ACTION act_Macinatore:
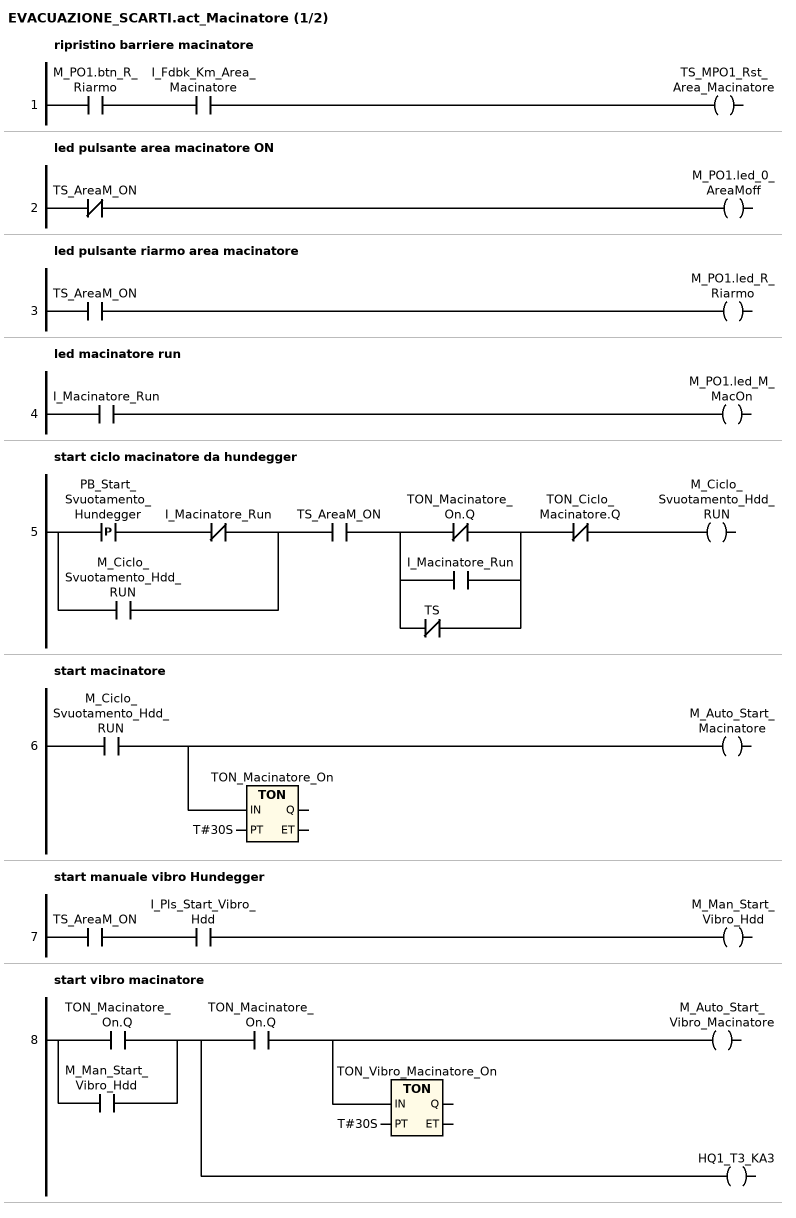
// NETWORK 1: ripristino barriere macinatore
TS_MPO1_Rst_Area_Macinatore := M_PO1.btn_R_Riarmo AND I_Fdbk_Km_Area_Macinatore;

// NETWORK 2: led pulsante area macinatore ON
M_PO1.led_0_AreaMoff := NOT TS_AreaM_ON;

// NETWORK 3: led pulsante riarmo area macinatore
M_PO1.led_R_Riarmo := TS_AreaM_ON;

// NETWORK 4: led macinatore run
M_PO1.led_M_MacOn := I_Macinatore_Run;

// NETWORK 5: start ciclo macinatore da hundegger
_rt1(CLK := PB_Start_Svuotamento_Hundegger);
M_Ciclo_Svuotamento_Hdd_RUN := (_rt1.Q AND NOT I_Macinatore_Run OR M_Ciclo_Svuotamento_Hdd_RUN) AND TS_AreaM_ON AND (NOT TON_Macinatore_On.Q OR I_Macinatore_Run OR NOT TS) AND NOT TON_Ciclo_Macinatore.Q;

// NETWORK 6: start macinatore
M_Auto_Start_Macinatore := M_Ciclo_Svuotamento_Hdd_RUN;
TON_Macinatore_On(IN := M_Ciclo_Svuotamento_Hdd_RUN, PT := T#30S); // TON

// NETWORK 7: start manuale vibro Hundegger
M_Man_Start_Vibro_Hdd := TS_AreaM_ON AND I_Pls_Start_Vibro_Hdd;

// NETWORK 8: start vibro macinatore
_w1 := TON_Macinatore_On.Q OR M_Man_Start_Vibro_Hdd;
_w2 := _w1 AND TON_Macinatore_On.Q;
M_Auto_Start_Vibro_Macinatore := _w2;
TON_Vibro_Macinatore_On(IN := _w2, PT := T#30S); // TON
HQ1_T3_KA3 := _w1;

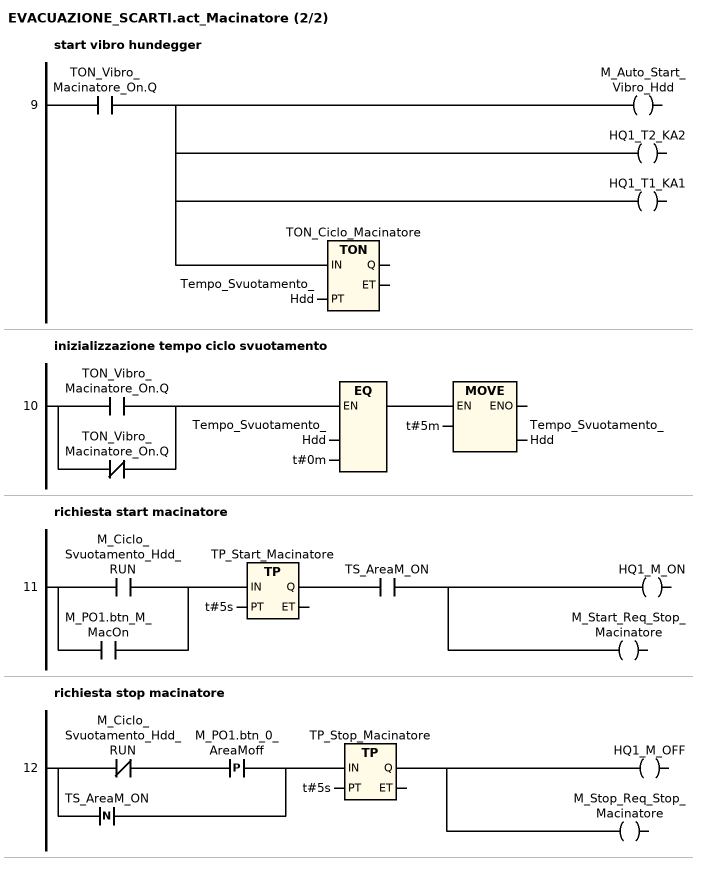
// NETWORK 9: start vibro hundegger
M_Auto_Start_Vibro_Hdd := TON_Vibro_Macinatore_On.Q;
HQ1_T2_KA2 := TON_Vibro_Macinatore_On.Q;
HQ1_T1_KA1 := TON_Vibro_Macinatore_On.Q;
TON_Ciclo_Macinatore(IN := TON_Vibro_Macinatore_On.Q, PT := Tempo_Svuotamento_Hdd); // TON

// NETWORK 10: inizializzazione tempo ciclo svuotamento
IF (TON_Vibro_Macinatore_On.Q OR NOT TON_Vibro_Macinatore_On.Q) AND Tempo_Svuotamento_Hdd = t#0m THEN
    Tempo_Svuotamento_Hdd := t#5m;
END_IF

// NETWORK 11: richiesta start macinatore
TP_Start_Macinatore(IN := M_Ciclo_Svuotamento_Hdd_RUN OR M_PO1.btn_M_MacOn, PT := t#5s); // TP
_w3 := TP_Start_Macinatore.Q AND TS_AreaM_ON;
HQ1_M_ON := _w3;
M_Start_Req_Stop_Macinatore := _w3;

// NETWORK 12: richiesta stop macinatore
_rt2(CLK := M_PO1.btn_0_AreaMoff);
_ft1(CLK := TS_AreaM_ON);
TP_Stop_Macinatore(IN := NOT M_Ciclo_Svuotamento_Hdd_RUN AND _rt2.Q OR _ft1.Q, PT := t#5s); // TP
HQ1_M_OFF := TP_Stop_Macinatore.Q;
M_Stop_Req_Stop_Macinatore := TP_Stop_Macinatore.Q;
END_ACTION

ACTION act_OUTPUT:

IF NOT bSIMULA_out THEN
	
	//TERM9 EL2008 H-Q1
	glo_dig_out_HQ1[1]		:=	Dis_Scarico_Hundegger;//S1_U1;									//DIGOUT CH1		Valvola aria pulizia ingresso M12
	glo_dig_out_HQ1[2]		:=	HQ1_T1_KA1;								//DIGOUT CH2		T1 Vibrotrasp buca
	glo_dig_out_HQ1[3]		:=	HQ1_T2_KA2;								//DIGOUT CH3		T2 Nastro elev buca
	glo_dig_out_HQ1[4]		:=	HQ1_T3_KA3;// AND NOT SensInMac;			//DIGOUT CH4		T3 Vibrotrasp macinatore
	glo_dig_out_HQ1[5]		:=	HQ1_T5M2_A_KA4;							//DIGOUT CH5		Apre scarico trasp orizz
	glo_dig_out_HQ1[6]		:=	HQ1_T5_KA5;								//DIGOUT CH6		Trasp elevat a parete
	glo_dig_out_HQ1[7]		:=	HQ1_T6_KA6;								//DIGOUT CH7		Trasp orizza a parete
	glo_dig_out_HQ1[8]		:=	HQ1_T5M2_C_KA7;							//DIGOUT CH8		Chiude scarico trasp orizz
	
	//TERM10 EL2008 H-Q1
	glo_dig_out_HQ1[9]		:= HQ1_T7_A_KA8;							//DIGOUT CH1		Caricatore macinat Avanti
	glo_dig_out_HQ1[10]		:= HQ1_T7_I_KA9;							//DIGOUT CH2		Caricatore macinat Indietro
	glo_dig_out_HQ1[11]		:= HQ1_M_ON;								//DIGOUT CH3		Macinatore ON impulsivo
	glo_dig_out_HQ1[12]		:= HQ1_M_OFF;								//DIGOUT CH4		Macinatore OFF impulsivo
	glo_dig_out_HQ1[13]		:= HQ1_T4_KA4;								//DIGOUT CH5		T4 Trasportatore silos macinatore	
	glo_dig_out_HQ1[14]		:= HQ1_S1_ValvolaStellare;					//DIGOUT CH6		Valvola stellare scarico silos 1	
	glo_dig_out_HQ1[15]		:= HQ1_RaclaON;								//DIGOUT CH7		Rancia: avviata da quadro silos
	glo_dig_out_HQ1[16]		:= HQ1_BrichettatriceON;					//DIGOUT CH8		Bricchettatrice: avviata da quadro silos

	//M_PO1											
	//IOLINK CH4		PULSANTIERA BNI005M
	glo_dig_out_T3C01[5] 	:= M_PO1.led_M_MacOn;						//BOTTONE '0'
	glo_dig_out_T3C01[8]	:= M_PO1.led_R_Riarmo;						//BOTTONE 'r'
	glo_dig_out_T3C01[6]	:= M_PO1.led_0_AreaMoff;					//TASTO 'M'
	
	//S1_PO1											
	//IOLINK CH4		PULSANTIERA BNI005M
					//BOTTONE 'r'

END_IF
END_ACTION

ACTION act_Semafori:

//#######################################################
//####################    SEMAFORI   ####################
//#######################################################

IF TS_AreaM_ON THEN
	IF I_Macinatore_Run  THEN
		fbS1_Se1(bON:= TRUE, sColore:= 3, bBlink:= TRUE, semaforo=> S1_Se1);	//verde	
	ELSE
		fbS1_Se1(bON:= TRUE, sColore:= 4, bBlink:= TRUE, semaforo=> S1_Se1);	//arancio
	END_IF
ELSE	
	fbS1_Se1(bON:= TRUE, sColore:= 2, bBlink:= TRUE, semaforo=> S1_Se1);	//rosso
END_IF
END_ACTION

ACTION act_Sensori:

//#######################################################
//####################    SENSORI   #####################
//#######################################################
//SOTTO HUNDEGGER
//CODA CIRCOLARE VALORI SENSORE inbit
T1SO1tmravg(IN:=TRUE,PT:=T#200MS);
T1SO1maxCnt:= REAL_TO_INT(T1SO1maxTimeavg*1000/200);
IF T1SO1maxCnt > 99 THEN
	T1SO1maxCnt:=99;
END_IF
IF T1SO1tmravg.Q THEN
	T1SO1tmravg(IN:=FALSE);	
	//CONTATORE TEMPO MASSIMO CAMPIONATURA
	IF T1SO1cnt < T1SO1maxCnt-1 THEN
		T1SO1cnt:=T1SO1cnt+1;	
	ELSE
		T1SO1cnt:=0;
	END_IF
	//POPOLO ARRAY LETTURE SENSORE in bit			
	T1SO1arravg[T1SO1cnt]:= T1_SO1;
END_IF
//MEDIA VALORI inbit
T1SO1cnt3:=0;
T1SO1sumavg:=0;
FOR T1SO1cnt2:=1 TO T1SO1maxCnt-1 DO
	IF T1SO1arravg[T1SO1cnt2] > 0 THEN
		T1SO1sumavg:= T1SO1sumavg + T1SO1arravg[T1SO1cnt2];
		T1SO1cnt3:=T1SO1cnt3+1;
	END_IF
END_FOR
IF T1SO1sumavg > 0 THEN
	T1SO1avg:=(T1SO1sumavg/T1SO1cnt3);	
END_IF
T1.SO1_fb(
	lettura:= REAL_TO_INT(T1SO1avg), 
	distanzaAVuoto:=6150,
	valSoglia:= solgiaT1SO1, 
	filtertime:=0,
	full=> appT1S01_Full);		
	
	//T1S01 full ritardato di 10 secondi 
	tmrT1S01_Full(IN:=appT1S01_Full,PT:=T#10S);
	T1.SO1_full := tmrT1S01_Full.Q;
	
//INGRESSO al T3
//CODA CIRCOLARE VALORI SENSORE inbit
T3S1tmravg(IN:=TRUE,PT:=T#200MS);
T3S1maxCnt:= REAL_TO_INT(T3S1maxTimeavg*1000/200);
IF T3S1maxCnt > 99 THEN
	T3S1maxCnt:=99;
END_IF
IF T3S1tmravg.Q THEN
	T3S1tmravg(IN:=FALSE);	
	//CONTATORE TEMPO MASSIMO CAMPIONATURA
	IF T3S1cnt < T3S1maxCnt-1 THEN
		T3S1cnt:=T3S1cnt+1;	
	ELSE
		T3S1cnt:=0;
	END_IF
	//POPOLO ARRAY LETTURE SENSORE in bit			
	T3S1arravg[T3S1cnt]:= T3_S1;
END_IF
//MEDIA VALORI inbit
T3S1cnt3:=0;
T3S1sumavg:=0;
FOR T3S1cnt2:=1 TO T3S1maxCnt-1 DO
	IF T3S1arravg[T3S1cnt2] > 0 THEN
		T3S1sumavg:= T3S1sumavg + T3S1arravg[T3S1cnt2];
		T3S1cnt3:=T3S1cnt3+1;
	END_IF
END_FOR
IF T3S1sumavg > 0 THEN
	T3S1avg:=(T3S1sumavg/T3S1cnt3);	
END_IF
T3.S1_fb(
	lettura:= REAL_TO_INT(T3S1avg), 
	maxScaleBit:= 32767, 
	maxScaleIng:= 1300, 
	deltaLowLimit:= 30,
	distanzaAVuoto:=1173,
	valSoglia:= sogliaT3S1, 
	filterTime:=2,
	full=> T3.S1_full,
	actualVal=> T3.S1_actVal);


//USCITA al T3	
//CODA CIRCOLARE VALORI SENSORE inbit
T3S2tmravg(IN:=TRUE,PT:=T#200MS);
T3S2maxCnt:= REAL_TO_INT(T3S2maxTimeavg*1000/200);
IF T3S2maxCnt > 99 THEN
	T3S2maxCnt:=99;
END_IF
IF T3S2tmravg.Q THEN
	T3S2tmravg(IN:=FALSE);	
	//CONTATORE TEMPO MASSIMO CAMPIONATURA
	IF T3S2cnt < T3S2maxCnt-1 THEN
		T3S2cnt:=T3S2cnt+1;	
	ELSE
		T3S2cnt:=0;
	END_IF
	//POPOLO ARRAY LETTURE SENSORE in bit			
	T3S2arravg[T3S2cnt]:= T3_S2;
END_IF
//MEDIA VALORI inbit
T3S2cnt3:=0;
T3S2sumavg:=0;
FOR T3S2cnt2:=1 TO T3S2maxCnt-1 DO
	IF T3S2arravg[T3S2cnt2] > 0 THEN
		T3S2sumavg:= T3S2sumavg + T3S2arravg[T3S2cnt2];
		T3S2cnt3:=T3S2cnt3+1;
	END_IF
END_FOR
IF T3S2sumavg > 0 THEN
	T3S2avg:=(T3S2sumavg/T3S2cnt3);	
END_IF	
T3.S2_fb(
	lettura:= REAL_TO_INT(T3S2avg), 
	maxScaleBit:= 32767, 
	maxScaleIng:= 1300, 
	deltaLowLimit:= 30,
	distanzaAVuoto:=590,
	valSoglia:= sogliaT3S2, 
	filterTime:=2,
	full=> T3.S2_full,
	actualVal=> T3.S2_actVal);


	

//SILOS1	
//CODA CIRCOLARE VALORI SENSORE inbit
S1SO2tmravg(IN:=TRUE,PT:=T#200MS);
S1SO2maxCnt:= REAL_TO_INT(S1SO2maxTimeavg*1000/200);
IF S1SO2maxCnt > 99 THEN
	S1SO2maxCnt:=99;
END_IF
IF S1SO2tmravg.Q THEN
	S1SO2tmravg(IN:=FALSE);	
	//CONTATORE TEMPO MASSIMO CAMPIONATURA
	IF S1SO2cnt < S1SO2maxCnt-1 THEN
		S1SO2cnt:=S1SO2cnt+1;	
	ELSE
		S1SO2cnt:=0;
	END_IF
	//POPOLO ARRAY LETTURE SENSORE in bit			
	S1SO2arravg[S1SO2cnt]:= S1_SO2;
END_IF
//MEDIA VALORI inbit
S1SO2cnt3:=0;
S1SO2sumavg:=0;
FOR S1SO2cnt2:=1 TO S1SO2maxCnt-1 DO
	IF S1SO2arravg[S1SO2cnt2] > 0 THEN
		S1SO2sumavg:= S1SO2sumavg + S1SO2arravg[S1SO2cnt2];
		S1SO2cnt3:=S1SO2cnt3+1;
	END_IF
END_FOR
IF S1SO2sumavg > 0 THEN
	S1SO2avg:=(S1SO2sumavg/S1SO2cnt3);	
END_IF
(*
S1.SO2_fb(
	lettura:= REAL_TO_INT(S1SO2avg), 
	maxScaleBit:= 32767, 
	maxScaleIng:= 6000, 
	deltaLowLimit:= 30, 
	distanzaAVuoto:=3250,
	valSoglia:= sogliaS1SO2, 
	filterTime:=1,
	full=> SO2_full_curr, //S1.SO2_full,
	actualVal=>S1.SO2_actVal);
	
	
	tmrValidaSoglia_S02(IN:= SO2_full_curr, PT:=T#15S);
	IF tmrValidaSoglia_S02.Q THEN
		tmrValidaSoglia_S02(IN:= FALSE);
		S1.SO2_full:= TRUE;
	END_IF
	
	IF NOT SO2_full_curr THEN
		S1.SO2_full:= FALSE;
	END_IF
	*)
	
//sensore livello silos (sensore in basso)

tmrS1_T_Rit_Empty(IN:=S1_S1,PT:=T#15m);
	S1.SO2_full:= TRUE;//tmrS1_T_Rit_Empty.Q OR Forza_TT1S01_Full;
	
//x HMI
glo_ES_ActVal.S1_S02:=S1.SO2_actVal;
altMatS1SO2:= S1.SO2_fb.distanzaAVuoto - glo_ES_ActVal.S1_S02;		
IF altMatS1SO2 <0 THEN
	altMatS1SO2:=0;
END_IF			
	


//SILOS2
S2.S1_fb(
	lettura:= S2_S1, 
	maxScaleBit:= 32767, 
	maxScaleIng:= 6000, 
	deltaLowLimit:= 30, 
	distanzaAVuoto:=6000,
	valSoglia:= 2000, 
	full=> S2.S1_full,
	actualVal=>S2.S1_actVal);
END_ACTION

END_PROGRAM

// ---- POUs/EVACUAZIONE_SCARTI/FB/FB_Semaforo.TcPOU
FUNCTION_BLOCK FB_Semaforo
VAR_INPUT
	bON			:BOOL;
	sColore		:int;
	bBlink		:BOOL;
END_VAR
VAR_OUTPUT
	semaforo	:ES_SEMAFORO;
END_VAR
VAR
	_tmrBlink	:ton;
	_bAccesa	:BOOL;
END_VAR


//1: BLU
//2: VERDE
//4: ROSSO
//6: ARANCIO

semaforo.analog0:= 0;
semaforo.analog1:= 0;
semaforo.analog2:= 0;
semaforo.analog3:= 0;
semaforo.analog4:= 0;
semaforo.analog5:= 0;
		
IF bBlink THEN
	_tmrBlink(IN:= bON, PT:=T#1000MS);
	IF _tmrBlink.Q THEN
		_tmrBlink(IN:= FALSE);
		_bAccesa:= NOT _bAccesa;
	END_IF
ELSE
	_bAccesa:=TRUE;
END_IF
		
IF bON THEN

	CASE sColore OF
				
	1: //BLU:
		IF _bAccesa THEN
			semaforo.analog1:= 1;
		END_IF 
		
	2: //ROSSO:
		IF _bAccesa THEN
			semaforo.analog2:= 4;
		END_IF
		
	3: //VERDE:
		IF _bAccesa THEN
			semaforo.analog3:= 2;
		END_IF
		
	4: //ARANCIO:
		IF _bAccesa THEN
			semaforo.analog4:= 6;
		END_IF
				
	
	END_CASE


END_IF

END_FUNCTION_BLOCK

// ---- POUs/EVACUAZIONE_SCARTI/FB/fun_AreaM_SPEGNITUTTO.TcPOU
FUNCTION fun_AreaM_SPEGNITUTTO : FB_Semaforo
VAR_INPUT
END_VAR
VAR
	bT3EnTPausaLavoro: BOOL;
END_VAR


//bit di COMANDO (cmd nellinterfaccia)
bT1_ON:=FALSE;
bT2_ON:=FALSE;
bT3_ON:=FALSE;
T3_ModoPausaLavoro:=FALSE;
bT3EnT1PausaLavoro:=FALSE;
bT3EnT2PausaLavoro:=FALSE;
T3_Lavoro :=FALSE;	
M_Start_Macinatore_Loc := FALSE;
bT4_ON:=FALSE;
bM_ON:=FALSE;


bMacinatoreStop:=TRUE;
bMacinatoreStart:=FALSE;
bT3T5T6DelayStart:=FALSE;

//uscite finali
HQ1_T1_KA1:=FALSE;
HQ1_T2_KA2:=FALSE;
HQ1_T3_KA3:=FALSE;
HQ1_T4_KA4:=FALSE;
HQ1_T5_KA5:=FALSE;
HQ1_T6_KA6:=FALSE;

//macchine a stati
stepT1T2:=100;
stepT3:=100;
stepT4:=100;
descT1T2:='T1-T2 disabilitati';
descT3:='T3 disabilitati';
descT4:='T4 disabilitati';

END_FUNCTION

// ---- POUs/RULLI_CENTRO_TAGLI/MAIN_RCT.TcPOU
PROGRAM MAIN_RCT
VAR
END_VAR


RULLI_CENTRO_TAGLI();

END_PROGRAM

// ---- POUs/EVACUAZIONE_SCARTI/FB/FB_AnalogSensor_full.TcPOU
FUNCTION_BLOCK FB_AnalogSensor_full
VAR_INPUT
	lettura			:INT;
	maxScaleBit		:INT;
	maxScaleIng		:INT;
	deltaLowLimit	:INT;
	distanzaAVuoto	:INT;
	valSoglia		:INT;
	filterTime		:INT;		//seconds
END_VAR
VAR_OUTPUT
	full			:BOOL;
	actualVal		:INT;
END_VAR
VAR
	_actVal			:INT;
	_tmr			:TON;
	_over			:BOOL;
END_VAR


_actVal := ((lettura*maxScaleIng)/maxScaleBit) - deltaLowLimit;
actualVal:=_actVal ;
IF distanzaAVuoto - _actVal > valSoglia THEN
	_over := TRUE;
ELSE
	full:=FALSE;
END_IF

_tmr(IN:=_over, PT:=INT_TO_TIME(filterTime*1000));
IF _tmr.Q THEN
	_over:=FALSE;
	full:=TRUE;
END_IF

END_FUNCTION_BLOCK

// ---- POUs/EVACUAZIONE_SCARTI/FB/FB_MMSensor_full.TcPOU
FUNCTION_BLOCK FB_MMSensor_full
VAR_INPUT
		lettura			:INT;
		distanzaAVuoto	:INT; 
		valSoglia		:INT;
		filterTime		:INT;		//seconds
END_VAR
VAR_OUTPUT
		full			:BOOL;
END_VAR
VAR
		_tmr			:TON;
		_over			:BOOL;
END_VAR



IF lettura < valSoglia THEN
	_over := TRUE;
ELSE
	_over:=FALSE;
	full:=FALSE;
END_IF

_tmr(IN:=_over, PT:=INT_TO_TIME(filterTime*1000));
IF _tmr.Q THEN
	_over:=FALSE;
	full:=TRUE;
END_IF

END_FUNCTION_BLOCK

// ---- POUs/RULLI_CENTRO_TAGLI/FB/FB_In_Position.TcPOU
FUNCTION_BLOCK FB_In_Position
VAR_INPUT
	Act_Position	:LREAL;
	Target_Position	:LREAL;	
	Toll_Window		:LREAL;
END_VAR
VAR_OUTPUT
	Axe_In_Pos		:BOOL;

END_VAR
VAR
	_pos_window		:LREAL;
	_neg_window		:LREAL;

END_VAR


_pos_window := Target_Position + Toll_Window;
_neg_window := Target_Position - Toll_Window;

IF (Act_Position >= _neg_window) AND  (Act_Position <= _pos_window) THEN
	Axe_In_Pos := TRUE;
ELSE
	Axe_In_Pos:=FALSE;
END_IF

END_FUNCTION_BLOCK
